PROGRAM F11_InfeedConvQueueCtrl
VAR
	fbSequenceControl					: FB_SYSTEM_SeqControl;
	nSequenceStep					: INT;
	b00_Idle							: BOOL;
	b01_ScanBarcode					: BOOL;
	b20_Done							: BOOL;

	bScannerBusy						: BOOL;
	fbScanTimeout					: TON;

	rtrigScanBarcode					: R_TRIG;
	fbScanDelay						: TON;
	fbScannerCtrl						: FB_SCANNER_CameraSelect;

	sLastGoodOuterBarcode				: T_OUTER_Barcode;
	sLastManualOuterBarcode			: T_OUTER_Barcode;

	fbOuterAggregationEvaluation			: FB_SCANNER_Evaluation;
	fbInfeedConvAggregated				: FB_CTU32;

	fbAddConvQueue					: FB_CASE_AddOuterToInfeedQ;
	fbMasterListControl					: FB_CASE_MasterListControl;

	tofAggregationCameraOFFDelay 	: TOF;


	fbAverageScanTime					: FB_SYSTEM_AverageTimeDiff;
	fbPerformance1							: FB_Interval;
	fbPerformance2							: FB_Interval;
END_VAR
(*
VAR CONSTANT
	sOptions						: ST_SCANNER_Options := (eScannerType := E_MV_440SR_FULL, nImageBuffer := 1, nExpectedResp := 1);
END_VAR*)
VAR // added by the converter: edge detectors and wires of the graphical bodies
    _w1 : BOOL;
END_VAR

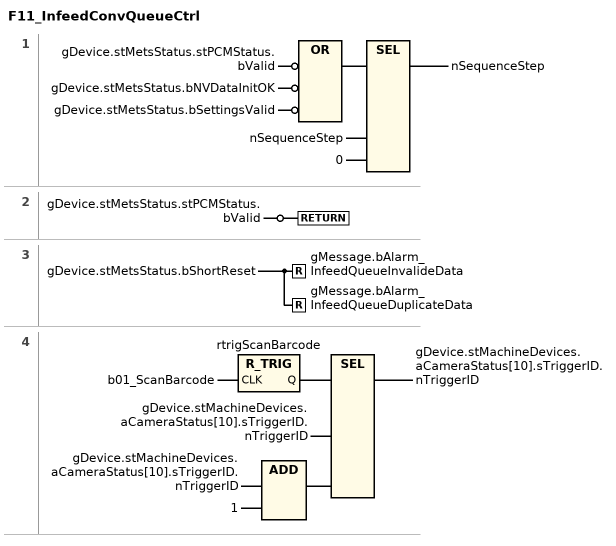
// NETWORK 1
nSequenceStep := SEL(NOT gDevice.stMetsStatus.stPCMStatus.bValid OR NOT gDevice.stMetsStatus.bNVDataInitOK OR NOT gDevice.stMetsStatus.bSettingsValid, nSequenceStep, 0);

// NETWORK 2
IF NOT gDevice.stMetsStatus.stPCMStatus.bValid THEN RETURN; END_IF

// NETWORK 3
gMessage.bAlarm_InfeedQueueInvalideData R= gDevice.stMetsStatus.bShortReset;
gMessage.bAlarm_InfeedQueueDuplicateData R= gDevice.stMetsStatus.bShortReset;

// NETWORK 4
rtrigScanBarcode(CLK := b01_ScanBarcode); // R_TRIG
gDevice.stMachineDevices.aCameraStatus[10].sTriggerID.nTriggerID := SEL(rtrigScanBarcode.Q, gDevice.stMachineDevices.aCameraStatus[10].sTriggerID.nTriggerID, gDevice.stMachineDevices.aCameraStatus[10].sTriggerID.nTriggerID + 1);

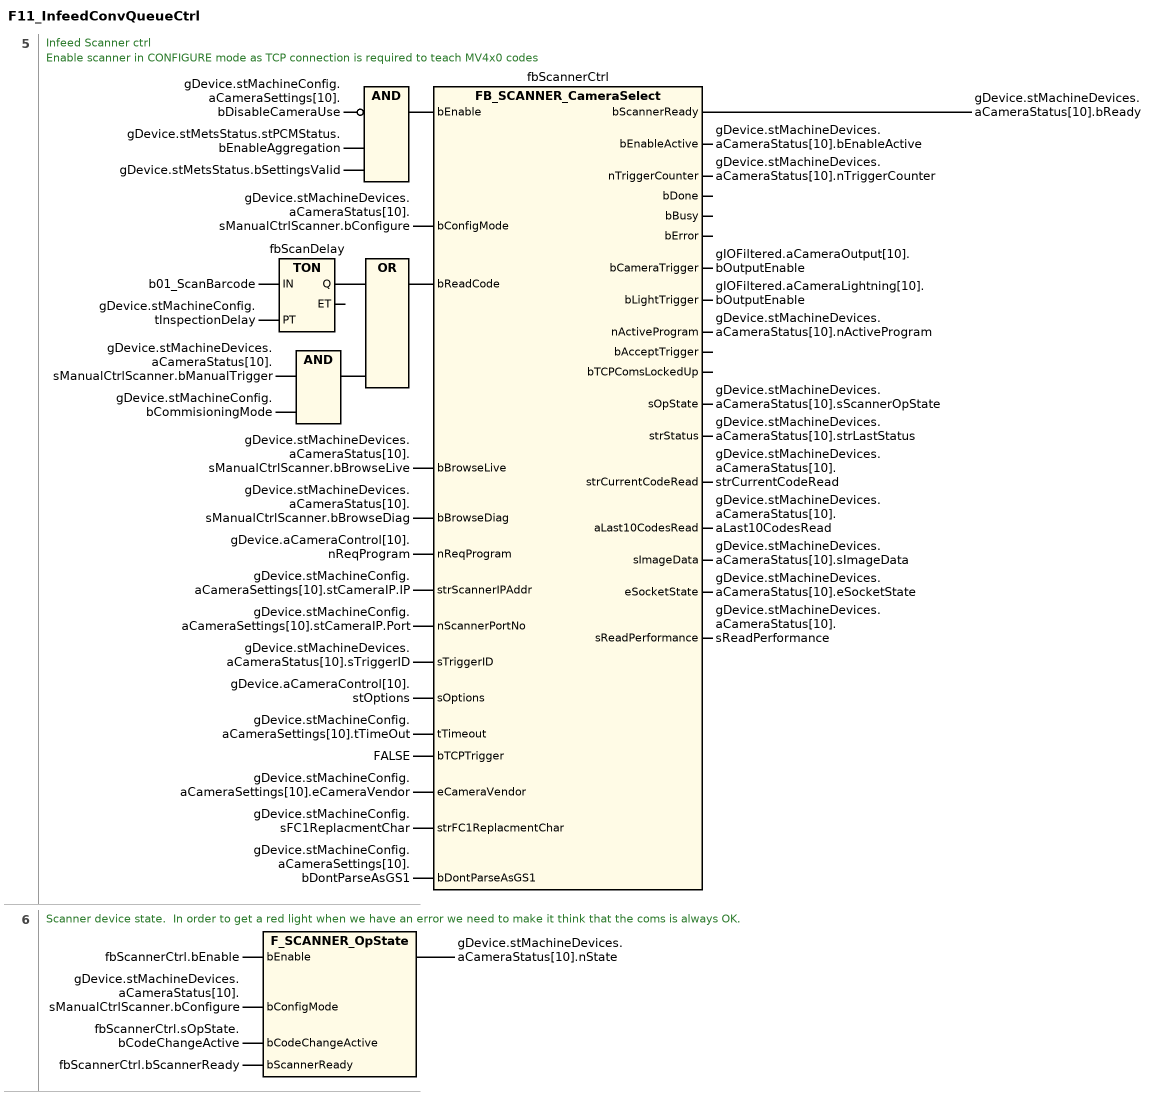
// NETWORK 5
// 					Infeed Scanner ctrl
// Enable scanner in CONFIGURE mode as TCP connection is required to teach MV4x0 codes
//
fbScanDelay(IN := b01_ScanBarcode, PT := gDevice.stMachineConfig.tInspectionDelay); // TON
fbScannerCtrl(
    bEnable := NOT gDevice.stMachineConfig.aCameraSettings[10].bDisableCameraUse AND gDevice.stMetsStatus.stPCMStatus.bEnableAggregation AND gDevice.stMetsStatus.bSettingsValid,
    bConfigMode := gDevice.stMachineDevices.aCameraStatus[10].sManualCtrlScanner.bConfigure,
    bReadCode := fbScanDelay.Q OR gDevice.stMachineDevices.aCameraStatus[10].sManualCtrlScanner.bManualTrigger AND gDevice.stMachineConfig.bCommisioningMode,
    bBrowseLive := gDevice.stMachineDevices.aCameraStatus[10].sManualCtrlScanner.bBrowseLive,
    bBrowseDiag := gDevice.stMachineDevices.aCameraStatus[10].sManualCtrlScanner.bBrowseDiag,
    nReqProgram := gDevice.aCameraControl[10].nReqProgram,
    strScannerIPAddr := gDevice.stMachineConfig.aCameraSettings[10].stCameraIP.IP,
    nScannerPortNo := gDevice.stMachineConfig.aCameraSettings[10].stCameraIP.Port,
    sTriggerID := gDevice.stMachineDevices.aCameraStatus[10].sTriggerID,
    sOptions := gDevice.aCameraControl[10].stOptions,
    tTimeout := gDevice.stMachineConfig.aCameraSettings[10].tTimeOut,
    bTCPTrigger := FALSE,
    eCameraVendor := gDevice.stMachineConfig.aCameraSettings[10].eCameraVendor,
    strFC1ReplacmentChar := gDevice.stMachineConfig.sFC1ReplacmentChar,
    bDontParseAsGS1 := gDevice.stMachineConfig.aCameraSettings[10].bDontParseAsGS1,
    bEnableActive => gDevice.stMachineDevices.aCameraStatus[10].bEnableActive,
    nTriggerCounter => gDevice.stMachineDevices.aCameraStatus[10].nTriggerCounter,
    bCameraTrigger => gIOFiltered.aCameraOutput[10].bOutputEnable,
    bLightTrigger => gIOFiltered.aCameraLightning[10].bOutputEnable,
    nActiveProgram => gDevice.stMachineDevices.aCameraStatus[10].nActiveProgram,
    sOpState => gDevice.stMachineDevices.aCameraStatus[10].sScannerOpState,
    strStatus => gDevice.stMachineDevices.aCameraStatus[10].strLastStatus,
    strCurrentCodeRead => gDevice.stMachineDevices.aCameraStatus[10].strCurrentCodeRead,
    aLast10CodesRead => gDevice.stMachineDevices.aCameraStatus[10].aLast10CodesRead,
    sImageData => gDevice.stMachineDevices.aCameraStatus[10].sImageData,
    eSocketState => gDevice.stMachineDevices.aCameraStatus[10].eSocketState,
    sReadPerformance => gDevice.stMachineDevices.aCameraStatus[10].sReadPerformance); // FB_SCANNER_CameraSelect
gDevice.stMachineDevices.aCameraStatus[10].bReady := fbScannerCtrl.bScannerReady;

// NETWORK 6
// Scanner device state.  In order to get a red light when we have an error we need to make it think that the coms is always OK.
gDevice.stMachineDevices.aCameraStatus[10].nState := F_SCANNER_OpState(bEnable := fbScannerCtrl.bEnable, bConfigMode := gDevice.stMachineDevices.aCameraStatus[10].sManualCtrlScanner.bConfigure, bCodeChangeActive := fbScannerCtrl.sOpState.bCodeChangeActive, bScannerReady := fbScannerCtrl.bScannerReady);

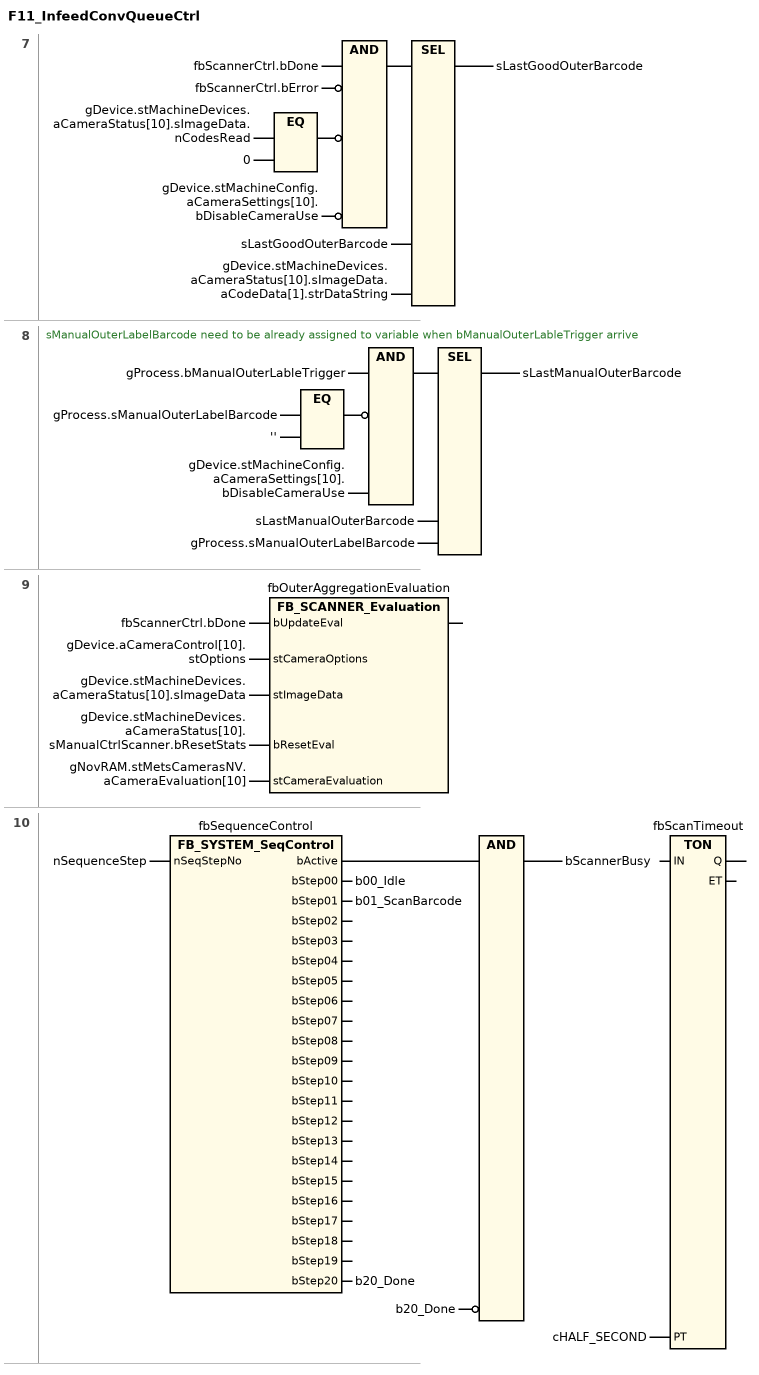
// NETWORK 7
sLastGoodOuterBarcode := SEL(fbScannerCtrl.bDone AND NOT fbScannerCtrl.bError AND NOT (gDevice.stMachineDevices.aCameraStatus[10].sImageData.nCodesRead = 0) AND NOT gDevice.stMachineConfig.aCameraSettings[10].bDisableCameraUse, sLastGoodOuterBarcode, gDevice.stMachineDevices.aCameraStatus[10].sImageData.aCodeData[1].strDataString);

// NETWORK 8
// sManualOuterLabelBarcode need to be already assigned to variable when bManualOuterLableTrigger arrive
sLastManualOuterBarcode := SEL(gProcess.bManualOuterLableTrigger AND NOT (gProcess.sManualOuterLabelBarcode = '') AND gDevice.stMachineConfig.aCameraSettings[10].bDisableCameraUse, sLastManualOuterBarcode, gProcess.sManualOuterLabelBarcode);

// NETWORK 9
fbOuterAggregationEvaluation(
    bUpdateEval := fbScannerCtrl.bDone,
    stCameraOptions := gDevice.aCameraControl[10].stOptions,
    stImageData := gDevice.stMachineDevices.aCameraStatus[10].sImageData,
    bResetEval := gDevice.stMachineDevices.aCameraStatus[10].sManualCtrlScanner.bResetStats,
    stCameraEvaluation := gNovRAM.stMetsCamerasNV.aCameraEvaluation[10]); // FB_SCANNER_Evaluation

// NETWORK 10
fbSequenceControl(
    nSeqStepNo := nSequenceStep,
    bStep00 => b00_Idle,
    bStep01 => b01_ScanBarcode,
    bStep20 => b20_Done); // FB_SYSTEM_SeqControl
_w1 := fbSequenceControl.bActive AND NOT b20_Done;
bScannerBusy := _w1;
fbScanTimeout(IN := _w1, PT := cHALF_SECOND); // TON

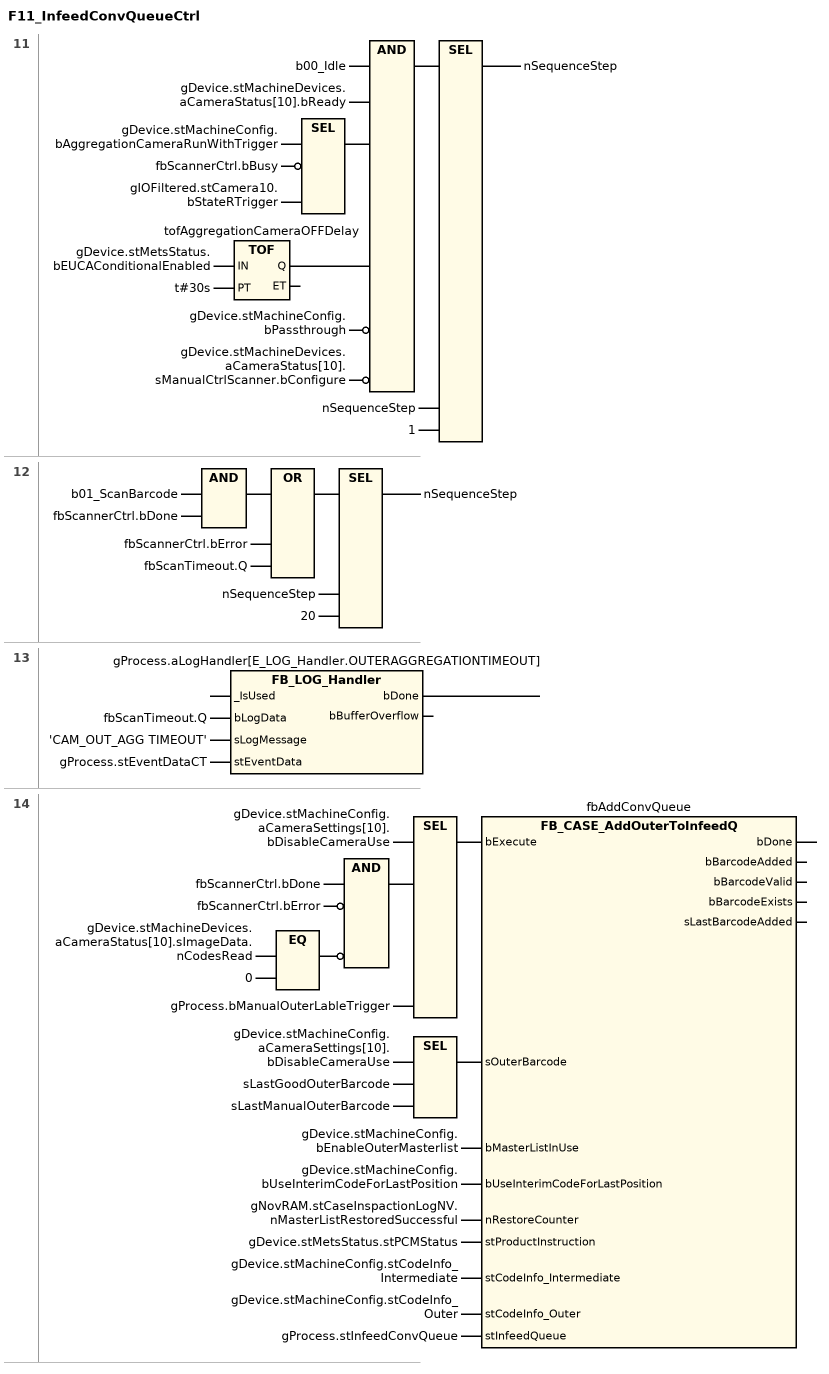
// NETWORK 11
tofAggregationCameraOFFDelay(IN := gDevice.stMetsStatus.bEUCAConditionalEnabled, PT := t#30s); // TOF
nSequenceStep := SEL(b00_Idle AND gDevice.stMachineDevices.aCameraStatus[10].bReady AND SEL(gDevice.stMachineConfig.bAggregationCameraRunWithTrigger, NOT fbScannerCtrl.bBusy, gIOFiltered.stCamera10.bStateRTrigger) AND tofAggregationCameraOFFDelay.Q AND NOT gDevice.stMachineConfig.bPassthrough AND NOT gDevice.stMachineDevices.aCameraStatus[10].sManualCtrlScanner.bConfigure, nSequenceStep, 1);

// NETWORK 12
nSequenceStep := SEL(b01_ScanBarcode AND fbScannerCtrl.bDone OR fbScannerCtrl.bError OR fbScanTimeout.Q, nSequenceStep, 20);

// NETWORK 13
gProcess.aLogHandler[E_LOG_Handler.OUTERAGGREGATIONTIMEOUT](
    bLogData := fbScanTimeout.Q,
    sLogMessage := 'CAM_OUT_AGG TIMEOUT',
    stEventData := gProcess.stEventDataCT); // FB_LOG_Handler

// NETWORK 14
fbAddConvQueue(
    bExecute := SEL(gDevice.stMachineConfig.aCameraSettings[10].bDisableCameraUse, fbScannerCtrl.bDone AND NOT fbScannerCtrl.bError AND NOT (gDevice.stMachineDevices.aCameraStatus[10].sImageData.nCodesRead = 0), gProcess.bManualOuterLableTrigger),
    sOuterBarcode := SEL(gDevice.stMachineConfig.aCameraSettings[10].bDisableCameraUse, sLastGoodOuterBarcode, sLastManualOuterBarcode),
    bMasterListInUse := gDevice.stMachineConfig.bEnableOuterMasterlist,
    bUseInterimCodeForLastPosition := gDevice.stMachineConfig.bUseInterimCodeForLastPosition,
    nRestoreCounter := gNovRAM.stCaseInspactionLogNV.nMasterListRestoredSuccessful,
    stProductInstruction := gDevice.stMetsStatus.stPCMStatus,
    stCodeInfo_Intermediate := gDevice.stMachineConfig.stCodeInfo_Intermediate,
    stCodeInfo_Outer := gDevice.stMachineConfig.stCodeInfo_Outer,
    stInfeedQueue := gProcess.stInfeedConvQueue); // FB_CASE_AddOuterToInfeedQ

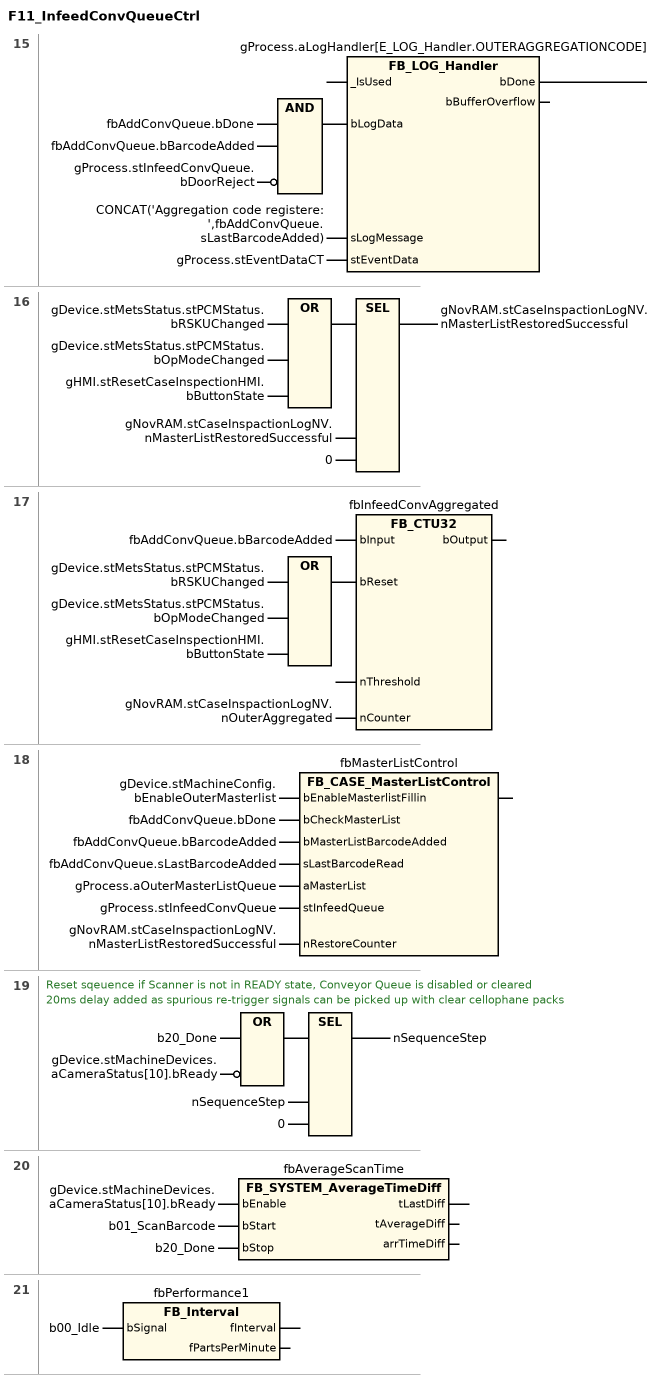
// NETWORK 15
gProcess.aLogHandler[E_LOG_Handler.OUTERAGGREGATIONCODE](
    bLogData := fbAddConvQueue.bDone AND fbAddConvQueue.bBarcodeAdded AND NOT gProcess.stInfeedConvQueue.bDoorReject,
    sLogMessage := CONCAT('Aggregation code registere: ',fbAddConvQueue.sLastBarcodeAdded),
    stEventData := gProcess.stEventDataCT); // FB_LOG_Handler

// NETWORK 16
gNovRAM.stCaseInspactionLogNV.nMasterListRestoredSuccessful := SEL(gDevice.stMetsStatus.stPCMStatus.bRSKUChanged OR gDevice.stMetsStatus.stPCMStatus.bOpModeChanged OR gHMI.stResetCaseInspectionHMI.bButtonState, gNovRAM.stCaseInspactionLogNV.nMasterListRestoredSuccessful, 0);

// NETWORK 17
fbInfeedConvAggregated(
    bInput := fbAddConvQueue.bBarcodeAdded,
    bReset := gDevice.stMetsStatus.stPCMStatus.bRSKUChanged OR gDevice.stMetsStatus.stPCMStatus.bOpModeChanged OR gHMI.stResetCaseInspectionHMI.bButtonState,
    nCounter := gNovRAM.stCaseInspactionLogNV.nOuterAggregated); // FB_CTU32

// NETWORK 18
fbMasterListControl(
    bEnableMasterlistFillin := gDevice.stMachineConfig.bEnableOuterMasterlist,
    bCheckMasterList := fbAddConvQueue.bDone,
    bMasterListBarcodeAdded := fbAddConvQueue.bBarcodeAdded,
    sLastBarcodeRead := fbAddConvQueue.sLastBarcodeAdded,
    aMasterList := gProcess.aOuterMasterListQueue,
    stInfeedQueue := gProcess.stInfeedConvQueue,
    nRestoreCounter := gNovRAM.stCaseInspactionLogNV.nMasterListRestoredSuccessful); // FB_CASE_MasterListControl

// NETWORK 19
// 					Reset sqeuence if Scanner is not in READY state, Conveyor Queue is disabled or cleared
// 20ms delay added as spurious re-trigger signals can be picked up with clear cellophane packs
//
nSequenceStep := SEL(b20_Done OR NOT gDevice.stMachineDevices.aCameraStatus[10].bReady, nSequenceStep, 0);

// NETWORK 20
fbAverageScanTime(
    bEnable := gDevice.stMachineDevices.aCameraStatus[10].bReady,
    bStart := b01_ScanBarcode,
    bStop := b20_Done); // FB_SYSTEM_AverageTimeDiff

// NETWORK 21
fbPerformance1(bSignal := b00_Idle); // FB_Interval

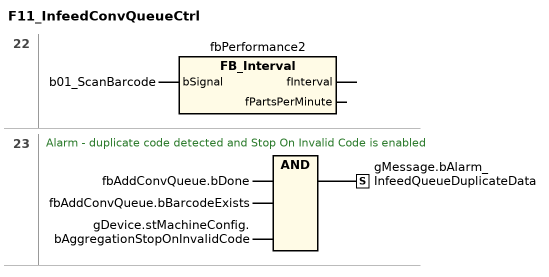
// NETWORK 22
fbPerformance2(bSignal := b01_ScanBarcode); // FB_Interval

// NETWORK 23
// Alarm - duplicate code detected and Stop On Invalid Code is enabled
gMessage.bAlarm_InfeedQueueDuplicateData S= fbAddConvQueue.bDone AND fbAddConvQueue.bBarcodeExists AND gDevice.stMachineConfig.bAggregationStopOnInvalidCode;

END_PROGRAM

(* stored: Version 1.1.0.1
   POU F11_InfeedConvQueueCtrl: Id {8da0d57e-1629-48e2-973d-ffd6029c3a89}, SpecialFunc None *)
